{attribute 'GeneratedUsingTerminal: EL2262-0000-0001'}
{attribute addProperty BoxType "EL2262-0000-0001"}
{attribute addProperty Id "WcStateAT %I*BOOL1"}
{attribute addProperty CRC "187373305"}
{attribute addProperty Size "1"}
TYPE WcState_0B2B16F9 :
STRUCT
	{attribute addProperty Name "WcState"}
	WcState AT %I* : BOOL;
END_STRUCT
END_TYPE

(* stored: Version 1.2.0.0, ProductVersion 3.1.4024.9
   DUT WcState_0B2B16F9: Id {baeaf054-e75f-4185-bb81-26e3f1dab17e} *)
